Fanuc KAREL source: ks00048.KL

-- PROVISIONAL review KL for V770-1; original PC SHA256 df6c27eac3cff046c6a02be0148d3228cd3fe8ae2f69fac752ff26ae6373f8fc
-- Incomplete behavior may be omitted. Consult companion uncertainty JSON. Do not deploy.
PROGRAM KS00048
%NOLOCKGROUP
BEGIN
  -- UNRESOLVED_PC offsets 5-13; opcodes 3F,75
  -- UNRESOLVED_PC offsets 18-27; opcodes 3F,75
  -- UNRESOLVED_PC offsets 32-70; opcodes 27,22,22,2A,22,2A,22,22,AF
  -- UNRESOLVED_PC offsets 75-79; opcodes 7F
END KS00048
